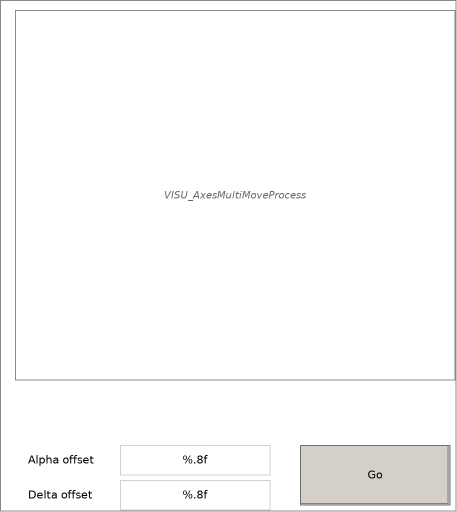
VISUALIZATION VISU_AxesManual_Offsets_OLD  // 457x512
VAR_IN_OUT
	ref : Axes;
    widget : AxesManualOffsetsWidget;
END_VAR
    Frame (15,10 440x370)
        shows VISU_AxesMultiMoveProcess(ref := ref.processes.moveRelative, widget := widget.moveRelative)
    Textfield (120,445 150x30), "%.8f", text variable: ref.processes.pointRelative.set.alpha
        OnMouseClick: write the text variable via VisuDialogs.Numpad
    Label (25,445 100x30), "Alpha offset"
    Textfield (120,480 150x30), "%.8f", text variable: ref.processes.pointRelative.set.delta
        OnMouseClick: write the text variable via VisuDialogs.Numpad
    Label (25,480 100x30), "Delta offset"
    Button (300,445 150x60), "Go", input disabled if: ref.processes.pointRelative.statuses.enabledStatus.disabled
        OnMouseClick: execute { ref.processes.pointRelative.do_request := TRUE; }
END_VISUALIZATION

(* stored: Version 1.1.0.1, ProductVersion 3.1.4019.2
   Visu VISU_AxesManual_Offsets_OLD: Id {63257011-6fac-4d70-ae7f-393247084915} *)
